// SIMATIC STEP 7 (V5.x) project timers&Counter
// CPU: CPU 313C
// station: Hardware
// station: SIMATIC 300(1)
// station: P_ADR_BUS
// program: S7 Program(1)

ORGANIZATION_BLOCK OB 1
TITLE = "Main Program Sweep (Cycle)"
VERSION : 0.1
VAR_TEMP
  OB1_EV_CLASS : BYTE ;	//Bits 0-3 = 1 (Coming event), Bits 4-7 = 1 (Event class 1)
  OB1_SCAN_1 : BYTE ;	//1 (Cold restart scan 1 of OB 1), 3 (Scan 2-n of OB 1)
  OB1_PRIORITY : BYTE ;	//Priority of OB Execution
  OB1_OB_NUMBR : BYTE ;	//1 (Organization block 1, OB1)
  OB1_RESERVED_1 : BYTE ;	//Reserved for system
  OB1_RESERVED_2 : BYTE ;	//Reserved for system
  OB1_PREV_CYCLE : INT ;	//Cycle time of previous OB1 scan (milliseconds)
  OB1_MIN_CYCLE : INT ;	//Minimum cycle time of OB1 (milliseconds)
  OB1_MAX_CYCLE : INT ;	//Maximum cycle time of OB1 (milliseconds)
  OB1_DATE_TIME : DATE_AND_TIME ;	//Date and time OB1 started
END_VAR
BEGIN
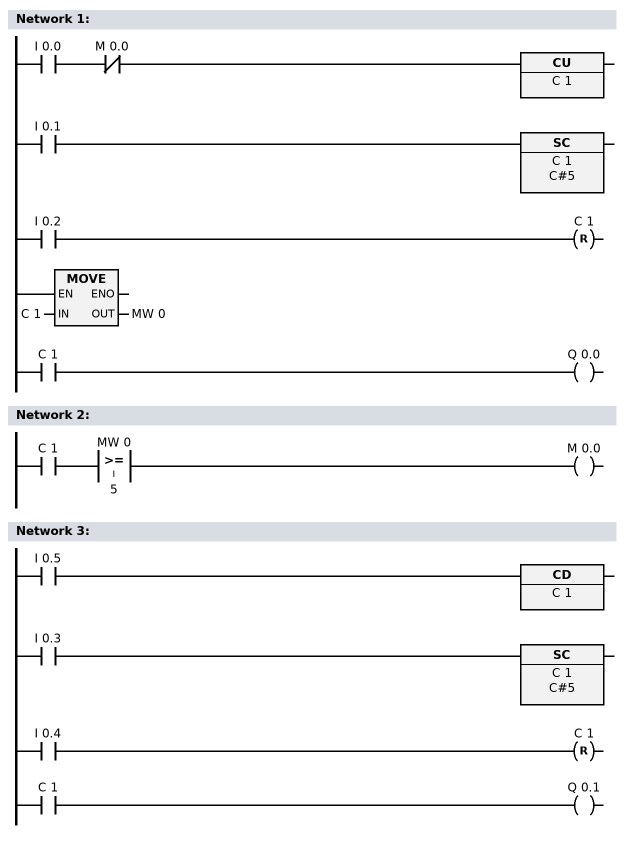
NETWORK
TITLE =
      A     I 0.0;
      AN    M 0.0;
      CU    C 1;
      BLD   101;
      A     I 0.1;
      L     C#5;
      S     C 1;
      A     I 0.2;
      R     C 1;
      L     C 1;
      T     MW 0;
      NOP   0;
      A     C 1;
      =     Q 0.0;
NETWORK
TITLE =
      A     C 1;
      A(;
      L     MW 0;
      L     5;
      >=I;
      );
      =     M 0.0;
NETWORK
TITLE =
      A     I 0.5;
      CD    C 1;
      BLD   101;
      A     I 0.3;
      L     C#5;
      S     C 1;
      A     I 0.4;
      R     C 1;
      NOP   0;
      NOP   0;
      A     C 1;
      =     Q 0.1;
END_ORGANIZATION_BLOCK
